// TIA Portal V18 export
FUNCTION "level Control" : Void   // FC20, LAD
{ S7_Optimized_Access := 'TRUE' }
VERSION : 0.1
// stored: AutoNumber true, IsIECCheckEnabled false, SetENOAutomatically false, UDAEnableTagReadback false
   VAR_TEMP   // added for the SCL form of the ladder/FBD networks
      _w1 : Bool;
   END_VAR
BEGIN

REGION Network 1: Level Sensor Tank A
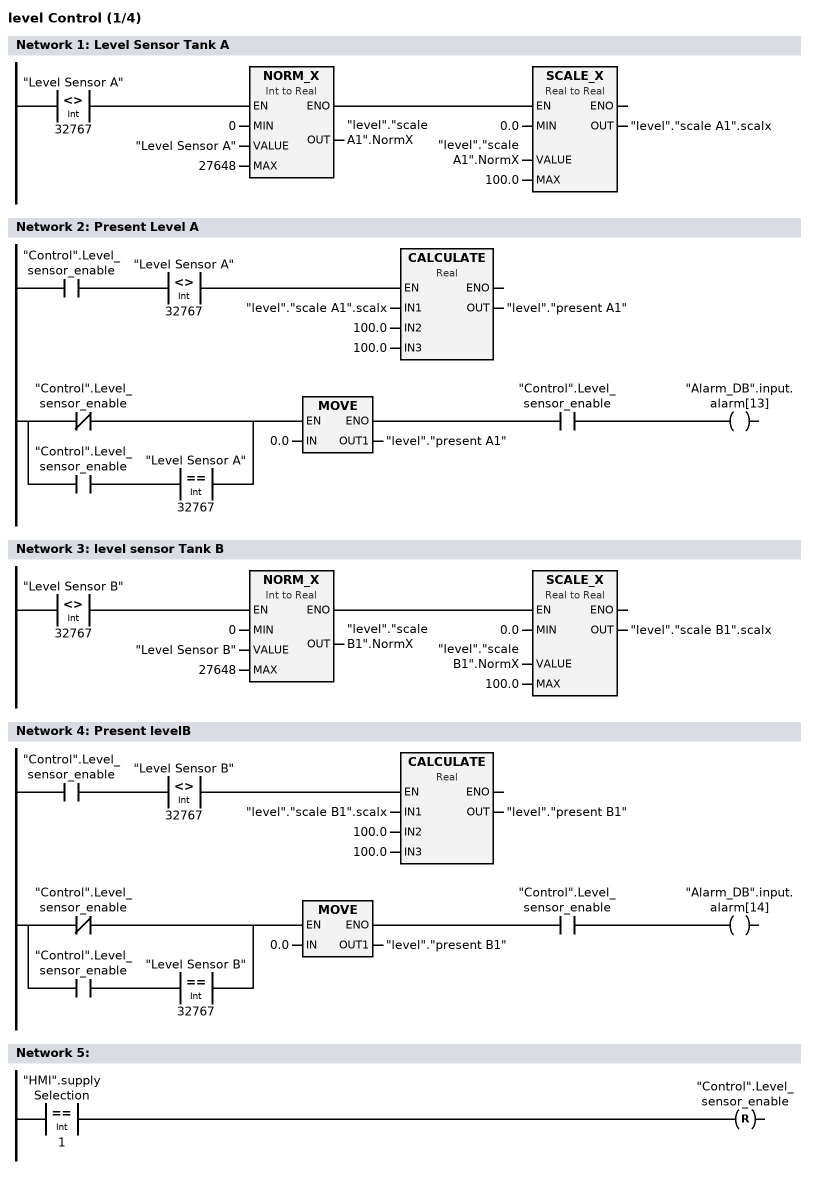
   RUNG wire#powerrail
      { S7_Templates := "SrcType := Int" } NE_Contact(in1 := "Level Sensor A", in2 := 32767)
      { S7_Templates := "[SrcType := Int, DestType := Real]" } Normalize(min := 0, value := "Level Sensor A", max := 27648, out => "level"."scale A1".NormX)
      { S7_Templates := "[SrcType := Real, DestType := Real]" } Scale(min := 0.0, value := "level"."scale A1".NormX, max := 100.0, out => "level"."scale A1".scalx)
   END_RUNG
   // the same network as SCL:
   IF "Level Sensor A" <> 32767 THEN
       "level"."scale A1".NormX := NORM_X(MIN := 0, VALUE := "Level Sensor A", MAX := 27648);
       "level"."scale A1".scalx := SCALE_X(MIN := 0.0, VALUE := "level"."scale A1".NormX, MAX := 100.0);
   END_IF;
END_REGION

REGION Network 2: Present Level A
   RUNG wire#powerrail
      Contact( "Control".Level_sensor_enable )
      { S7_Templates := "SrcType := Int" } NE_Contact(in1 := "Level Sensor A", in2 := 32767)
      { S7_Templates := "SrcType := Real"; S7_Expression := "ROUND(IN1*IN2)/IN3" } Calculate(in1 := "level"."scale A1".scalx, in2 := 100.0, in3 := 100.0, out => "level"."present A1")
   END_RUNG
   RUNG wire#powerrail
      I_Contact( "Control".Level_sensor_enable )
      wire#w1
      Move(in := 0.0, out1 => "level"."present A1")
      Contact( "Control".Level_sensor_enable )
      Coil( "Alarm_DB".input.alarm[13] )
   END_RUNG
   RUNG wire#powerrail
      Contact( "Control".Level_sensor_enable )
      { S7_Templates := "SrcType := Int" } EQ_Contact(in1 := "Level Sensor A", in2 := 32767)
   END_RUNG wire#w1
   // the same network as SCL:
   IF "Control".Level_sensor_enable AND ("Level Sensor A" <> 32767) THEN
       "level"."present A1" := ROUND("level"."scale A1".scalx*100.0)/100.0;
   END_IF;
   #_w1 := NOT "Control".Level_sensor_enable OR ("Control".Level_sensor_enable AND ("Level Sensor A" = 32767));
   IF #_w1 THEN "level"."present A1" := 0.0; END_IF;
   "Alarm_DB".input.alarm[13] := #_w1 AND "Control".Level_sensor_enable;
END_REGION

REGION Network 3: level sensor Tank B
   RUNG wire#powerrail
      { S7_Templates := "SrcType := Int" } NE_Contact(in1 := "Level Sensor B", in2 := 32767)
      { S7_Templates := "[SrcType := Int, DestType := Real]" } Normalize(min := 0, value := "Level Sensor B", max := 27648, out => "level"."scale B1".NormX)
      { S7_Templates := "[SrcType := Real, DestType := Real]" } Scale(min := 0.0, value := "level"."scale B1".NormX, max := 100.0, out => "level"."scale B1".scalx)
   END_RUNG
   // the same network as SCL:
   IF "Level Sensor B" <> 32767 THEN
       "level"."scale B1".NormX := NORM_X(MIN := 0, VALUE := "Level Sensor B", MAX := 27648);
       "level"."scale B1".scalx := SCALE_X(MIN := 0.0, VALUE := "level"."scale B1".NormX, MAX := 100.0);
   END_IF;
END_REGION

REGION Network 4: Present levelB
   RUNG wire#powerrail
      Contact( "Control".Level_sensor_enable )
      { S7_Templates := "SrcType := Int" } NE_Contact(in1 := "Level Sensor B", in2 := 32767)
      { S7_Templates := "SrcType := Real"; S7_Expression := "ROUND(IN1*IN2)/IN3" } Calculate(in1 := "level"."scale B1".scalx, in2 := 100.0, in3 := 100.0, out => "level"."present B1")
   END_RUNG
   RUNG wire#powerrail
      I_Contact( "Control".Level_sensor_enable )
      wire#w1
      Move(in := 0.0, out1 => "level"."present B1")
      Contact( "Control".Level_sensor_enable )
      Coil( "Alarm_DB".input.alarm[14] )
   END_RUNG
   RUNG wire#powerrail
      Contact( "Control".Level_sensor_enable )
      { S7_Templates := "SrcType := Int" } EQ_Contact(in1 := "Level Sensor B", in2 := 32767)
   END_RUNG wire#w1
   // the same network as SCL:
   IF "Control".Level_sensor_enable AND ("Level Sensor B" <> 32767) THEN
       "level"."present B1" := ROUND("level"."scale B1".scalx*100.0)/100.0;
   END_IF;
   #_w1 := NOT "Control".Level_sensor_enable OR ("Control".Level_sensor_enable AND ("Level Sensor B" = 32767));
   IF #_w1 THEN "level"."present B1" := 0.0; END_IF;
   "Alarm_DB".input.alarm[14] := #_w1 AND "Control".Level_sensor_enable;
END_REGION

REGION Network 5
   RUNG wire#powerrail
      { S7_Templates := "SrcType := Int" } EQ_Contact(in1 := "HMI".supplySelection, in2 := 1)
      R_Coil( "Control".Level_sensor_enable )
   END_RUNG
   // the same network as SCL:
   IF "HMI".supplySelection = 1 THEN "Control".Level_sensor_enable := FALSE; END_IF;
END_REGION

REGION Network 6: Low level A
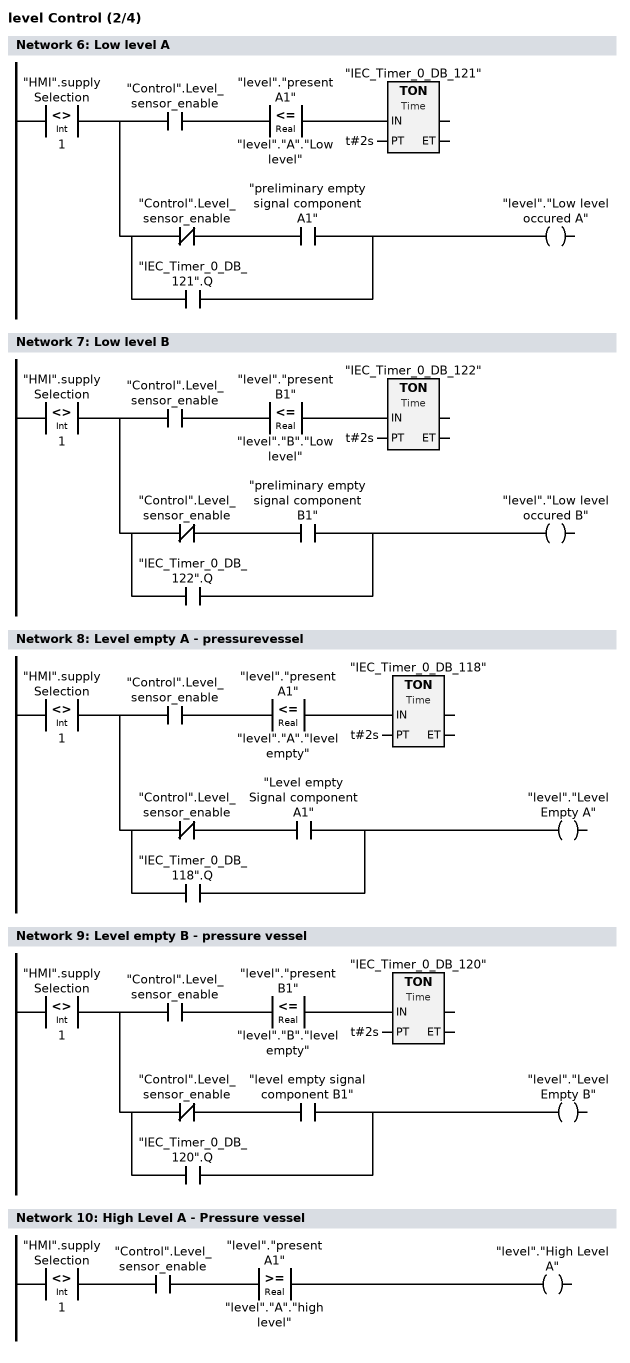
   RUNG wire#powerrail
      { S7_Templates := "SrcType := Int" } NE_Contact(in1 := "HMI".supplySelection, in2 := 1)
      wire#w1
      Contact( "Control".Level_sensor_enable )
      { S7_Templates := "SrcType := Real" } LE_Contact(in1 := "level"."present A1", in2 := "level"."A"."Low level")
      { S7_Templates := "time_type := Time" } "IEC_Timer_0_DB_121".TON(pt := t#2s, et =>)
   END_RUNG
   RUNG wire#w1
      I_Contact( "Control".Level_sensor_enable )
      Contact( "preliminary empty signal component A1" )
      wire#w2
      Coil( "level"."Low level occured A" )
   END_RUNG
   RUNG wire#w1
      Contact( "IEC_Timer_0_DB_121".Q )
   END_RUNG wire#w2
   // the same network as SCL:
   #_w1 := "HMI".supplySelection <> 1;
   "IEC_Timer_0_DB_121".TON(IN := #_w1 AND "Control".Level_sensor_enable AND ("level"."present A1" <= "level"."A"."Low level"),
                           PT := t#2s);
   "level"."Low level occured A" := #_w1 AND ((NOT "Control".Level_sensor_enable AND "preliminary empty signal component A1") OR "IEC_Timer_0_DB_121".Q);
END_REGION

REGION Network 7: Low level B
   RUNG wire#powerrail
      { S7_Templates := "SrcType := Int" } NE_Contact(in1 := "HMI".supplySelection, in2 := 1)
      wire#w1
      Contact( "Control".Level_sensor_enable )
      { S7_Templates := "SrcType := Real" } LE_Contact(in1 := "level"."present B1", in2 := "level"."B"."Low level")
      { S7_Templates := "time_type := Time" } "IEC_Timer_0_DB_122".TON(pt := t#2s, et =>)
   END_RUNG
   RUNG wire#w1
      I_Contact( "Control".Level_sensor_enable )
      Contact( "preliminary empty signal component B1" )
      wire#w2
      Coil( "level"."Low level occured B" )
   END_RUNG
   RUNG wire#w1
      Contact( "IEC_Timer_0_DB_122".Q )
   END_RUNG wire#w2
   // the same network as SCL:
   #_w1 := "HMI".supplySelection <> 1;
   "IEC_Timer_0_DB_122".TON(IN := #_w1 AND "Control".Level_sensor_enable AND ("level"."present B1" <= "level"."B"."Low level"),
                           PT := t#2s);
   "level"."Low level occured B" := #_w1 AND ((NOT "Control".Level_sensor_enable AND "preliminary empty signal component B1") OR "IEC_Timer_0_DB_122".Q);
END_REGION

REGION Network 8: Level empty A - pressurevessel
   RUNG wire#powerrail
      { S7_Templates := "SrcType := Int" } NE_Contact(in1 := "HMI".supplySelection, in2 := 1)
      wire#w1
      Contact( "Control".Level_sensor_enable )
      { S7_Templates := "SrcType := Real" } LE_Contact(in1 := "level"."present A1", in2 := "level"."A"."level empty")
      { S7_Templates := "time_type := Time" } "IEC_Timer_0_DB_118".TON(pt := t#2s, et =>)
   END_RUNG
   RUNG wire#w1
      I_Contact( "Control".Level_sensor_enable )
      Contact( "Level empty Signal component A1" )
      wire#w2
      Coil( "level"."Level Empty A" )
   END_RUNG
   RUNG wire#w1
      Contact( "IEC_Timer_0_DB_118".Q )
   END_RUNG wire#w2
   // the same network as SCL:
   #_w1 := "HMI".supplySelection <> 1;
   "IEC_Timer_0_DB_118".TON(IN := #_w1 AND "Control".Level_sensor_enable AND ("level"."present A1" <= "level"."A"."level empty"),
                           PT := t#2s);
   "level"."Level Empty A" := #_w1 AND ((NOT "Control".Level_sensor_enable AND "Level empty Signal component A1") OR "IEC_Timer_0_DB_118".Q);
END_REGION

REGION Network 9: Level empty B - pressure vessel
   RUNG wire#powerrail
      { S7_Templates := "SrcType := Int" } NE_Contact(in1 := "HMI".supplySelection, in2 := 1)
      wire#w1
      Contact( "Control".Level_sensor_enable )
      { S7_Templates := "SrcType := Real" } LE_Contact(in1 := "level"."present B1", in2 := "level"."B"."level empty")
      { S7_Templates := "time_type := Time" } "IEC_Timer_0_DB_120".TON(pt := t#2s, et =>)
   END_RUNG
   RUNG wire#w1
      I_Contact( "Control".Level_sensor_enable )
      Contact( "level empty signal component B1" )
      wire#w2
      Coil( "level"."Level Empty B" )
   END_RUNG
   RUNG wire#w1
      Contact( "IEC_Timer_0_DB_120".Q )
   END_RUNG wire#w2
   // the same network as SCL:
   #_w1 := "HMI".supplySelection <> 1;
   "IEC_Timer_0_DB_120".TON(IN := #_w1 AND "Control".Level_sensor_enable AND ("level"."present B1" <= "level"."B"."level empty"),
                           PT := t#2s);
   "level"."Level Empty B" := #_w1 AND ((NOT "Control".Level_sensor_enable AND "level empty signal component B1") OR "IEC_Timer_0_DB_120".Q);
END_REGION

REGION Network 10: High Level A - Pressure vessel
   RUNG wire#powerrail
      { S7_Templates := "SrcType := Int" } NE_Contact(in1 := "HMI".supplySelection, in2 := 1)
      Contact( "Control".Level_sensor_enable )
      { S7_Templates := "SrcType := Real" } GE_Contact(in1 := "level"."present A1", in2 := "level"."A"."high level")
      Coil( "level"."High Level A" )
   END_RUNG
   // the same network as SCL:
   "level"."High Level A" := ("HMI".supplySelection <> 1) AND "Control".Level_sensor_enable AND ("level"."present A1" >= "level"."A"."high level");
END_REGION

REGION Network 11: High Level B - Pressure Vessel
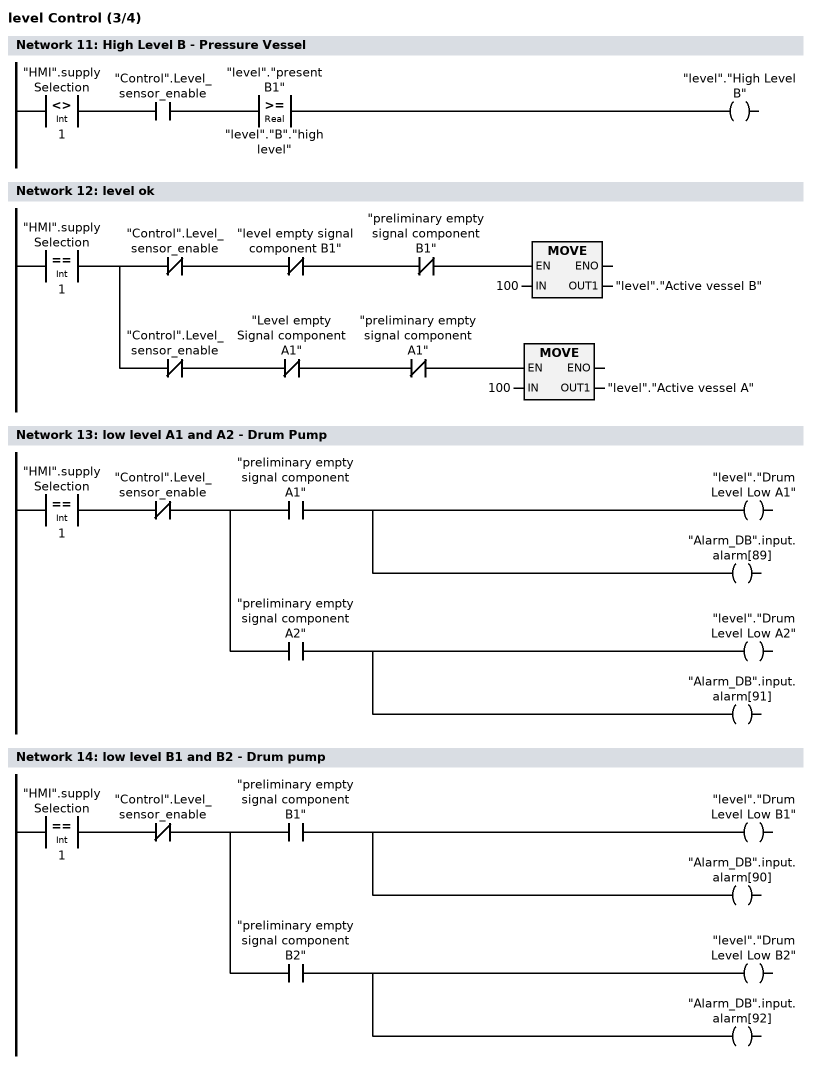
   RUNG wire#powerrail
      { S7_Templates := "SrcType := Int" } NE_Contact(in1 := "HMI".supplySelection, in2 := 1)
      Contact( "Control".Level_sensor_enable )
      { S7_Templates := "SrcType := Real" } GE_Contact(in1 := "level"."present B1", in2 := "level"."B"."high level")
      Coil( "level"."High Level B" )
   END_RUNG
   // the same network as SCL:
   "level"."High Level B" := ("HMI".supplySelection <> 1) AND "Control".Level_sensor_enable AND ("level"."present B1" >= "level"."B"."high level");
END_REGION

REGION Network 12: level ok
   RUNG wire#powerrail
      { S7_Templates := "SrcType := Int" } EQ_Contact(in1 := "HMI".supplySelection, in2 := 1)
      wire#w1
      I_Contact( "Control".Level_sensor_enable )
      I_Contact( "level empty signal component B1" )
      I_Contact( "preliminary empty signal component B1" )
      Move(in := 100, out1 => "level"."Active vessel B")
   END_RUNG
   RUNG wire#w1
      I_Contact( "Control".Level_sensor_enable )
      I_Contact( "Level empty Signal component A1" )
      I_Contact( "preliminary empty signal component A1" )
      Move(in := 100, out1 => "level"."Active vessel A")
   END_RUNG
   // the same network as SCL:
   #_w1 := "HMI".supplySelection = 1;
   IF #_w1 AND NOT "Control".Level_sensor_enable AND NOT "level empty signal component B1" AND NOT "preliminary empty signal component B1" THEN
       "level"."Active vessel B" := 100;
   END_IF;
   IF #_w1 AND NOT "Control".Level_sensor_enable AND NOT "Level empty Signal component A1" AND NOT "preliminary empty signal component A1" THEN
       "level"."Active vessel A" := 100;
   END_IF;
END_REGION

REGION Network 13: low level A1 and A2 - Drum Pump
   RUNG wire#powerrail
      { S7_Templates := "SrcType := Int" } EQ_Contact(in1 := "HMI".supplySelection, in2 := 1)
      I_Contact( "Control".Level_sensor_enable )
      wire#w1
      Contact( "preliminary empty signal component A1" )
      wire#w2
      Coil( "level"."Drum Level Low A1" )
   END_RUNG
   RUNG wire#w2
      Coil( "Alarm_DB".input.alarm[89] )
   END_RUNG
   RUNG wire#w1
      Contact( "preliminary empty signal component A2" )
      wire#w3
      Coil( "level"."Drum Level Low A2" )
   END_RUNG
   RUNG wire#w3
      Coil( "Alarm_DB".input.alarm[91] )
   END_RUNG
   // the same network as SCL:
   #_w1 := ("HMI".supplySelection = 1) AND NOT "Control".Level_sensor_enable;
   "level"."Drum Level Low A1" := #_w1 AND "preliminary empty signal component A1";
   "Alarm_DB".input.alarm[89] := "level"."Drum Level Low A1";
   "level"."Drum Level Low A2" := #_w1 AND "preliminary empty signal component A2";
   "Alarm_DB".input.alarm[91] := "level"."Drum Level Low A2";
END_REGION

REGION Network 14: low level B1 and B2 - Drum pump
   RUNG wire#powerrail
      { S7_Templates := "SrcType := Int" } EQ_Contact(in1 := "HMI".supplySelection, in2 := 1)
      I_Contact( "Control".Level_sensor_enable )
      wire#w1
      Contact( "preliminary empty signal component B1" )
      wire#w2
      Coil( "level"."Drum Level Low B1" )
   END_RUNG
   RUNG wire#w2
      Coil( "Alarm_DB".input.alarm[90] )
   END_RUNG
   RUNG wire#w1
      Contact( "preliminary empty signal component B2" )
      wire#w3
      Coil( "level"."Drum Level Low B2" )
   END_RUNG
   RUNG wire#w3
      Coil( "Alarm_DB".input.alarm[92] )
   END_RUNG
   // the same network as SCL:
   #_w1 := ("HMI".supplySelection = 1) AND NOT "Control".Level_sensor_enable;
   "level"."Drum Level Low B1" := #_w1 AND "preliminary empty signal component B1";
   "Alarm_DB".input.alarm[90] := "level"."Drum Level Low B1";
   "level"."Drum Level Low B2" := #_w1 AND "preliminary empty signal component B2";
   "Alarm_DB".input.alarm[92] := "level"."Drum Level Low B2";
END_REGION

REGION Network 15: level empty A1 and A2 - Drum pump
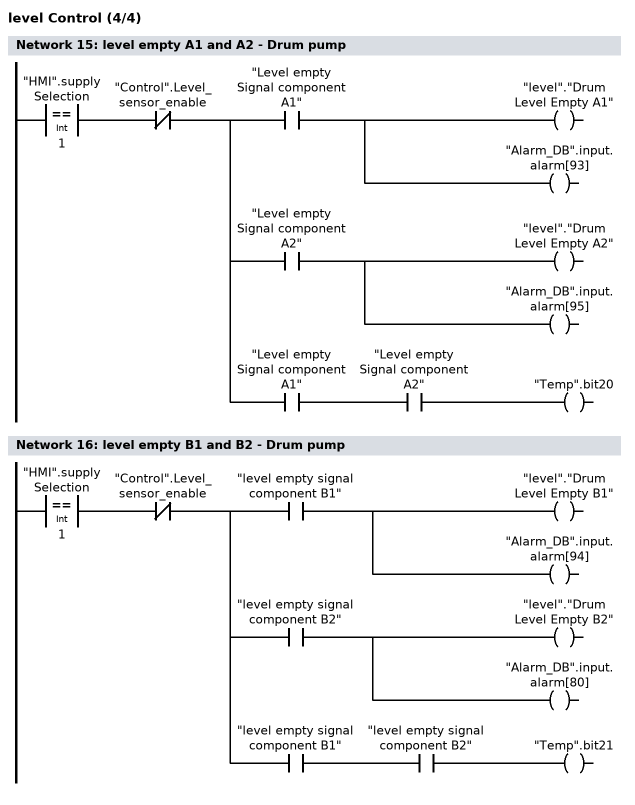
   RUNG wire#powerrail
      { S7_Templates := "SrcType := Int" } EQ_Contact(in1 := "HMI".supplySelection, in2 := 1)
      I_Contact( "Control".Level_sensor_enable )
      wire#w1
      Contact( "Level empty Signal component A1" )
      wire#w2
      Coil( "level"."Drum Level Empty A1" )
   END_RUNG
   RUNG wire#w2
      Coil( "Alarm_DB".input.alarm[93] )
   END_RUNG
   RUNG wire#w1
      Contact( "Level empty Signal component A2" )
      wire#w3
      Coil( "level"."Drum Level Empty A2" )
   END_RUNG
   RUNG wire#w3
      Coil( "Alarm_DB".input.alarm[95] )
   END_RUNG
   RUNG wire#w1
      Contact( "Level empty Signal component A1" )
      Contact( "Level empty Signal component A2" )
      Coil( "Temp".bit20 )
   END_RUNG
   // the same network as SCL:
   #_w1 := ("HMI".supplySelection = 1) AND NOT "Control".Level_sensor_enable;
   "level"."Drum Level Empty A1" := #_w1 AND "Level empty Signal component A1";
   "Alarm_DB".input.alarm[93] := "level"."Drum Level Empty A1";
   "level"."Drum Level Empty A2" := #_w1 AND "Level empty Signal component A2";
   "Alarm_DB".input.alarm[95] := "level"."Drum Level Empty A2";
   "Temp".bit20 := #_w1 AND "Level empty Signal component A1" AND "Level empty Signal component A2";
END_REGION

REGION Network 16: level empty B1 and B2 - Drum pump
   RUNG wire#powerrail
      { S7_Templates := "SrcType := Int" } EQ_Contact(in1 := "HMI".supplySelection, in2 := 1)
      I_Contact( "Control".Level_sensor_enable )
      wire#w1
      Contact( "level empty signal component B1" )
      wire#w2
      Coil( "level"."Drum Level Empty B1" )
   END_RUNG
   RUNG wire#w2
      Coil( "Alarm_DB".input.alarm[94] )
   END_RUNG
   RUNG wire#w1
      Contact( "level empty signal component B2" )
      wire#w3
      Coil( "level"."Drum Level Empty B2" )
   END_RUNG
   RUNG wire#w3
      Coil( "Alarm_DB".input.alarm[80] )
   END_RUNG
   RUNG wire#w1
      Contact( "level empty signal component B1" )
      Contact( "level empty signal component B2" )
      Coil( "Temp".bit21 )
   END_RUNG
   // the same network as SCL:
   #_w1 := ("HMI".supplySelection = 1) AND NOT "Control".Level_sensor_enable;
   "level"."Drum Level Empty B1" := #_w1 AND "level empty signal component B1";
   "Alarm_DB".input.alarm[94] := "level"."Drum Level Empty B1";
   "level"."Drum Level Empty B2" := #_w1 AND "level empty signal component B2";
   "Alarm_DB".input.alarm[80] := "level"."Drum Level Empty B2";
   "Temp".bit21 := #_w1 AND "level empty signal component B1" AND "level empty signal component B2";
END_REGION
END_FUNCTION
